FUNCTION_BLOCK FB_CintaTransferirPale_SFC
VAR_INPUT
    // SFC-Flags
    SFCPause: BOOL;
    SFCReset: BOOL;
    
    // Indicadores de sincronizacion
    Ack: BOOL := TRUE;
    Execute: BOOL;
    
    // Parametros
    TpoCintaRetenedor: TIME := T#1S;
    TpoCintaSeparador: TIME := T#1S;
    TpoPaleSalida: TIME := T#1S;
    TpoPaleTransferencia: TIME := T#1S;
    
    // Entradas
    PalePresencia: BOOL;
END_VAR
VAR_OUTPUT
    // Indicadores de sincronizacion
    Done: BOOL;
    Ready: BOOL;
    // Salidas
    CintaMotorActiva: BOOL;
    CintaRetenedorBaja: BOOL;
    CintaSeparadorSube: BOOL;
END_VAR
VAR
END_VAR

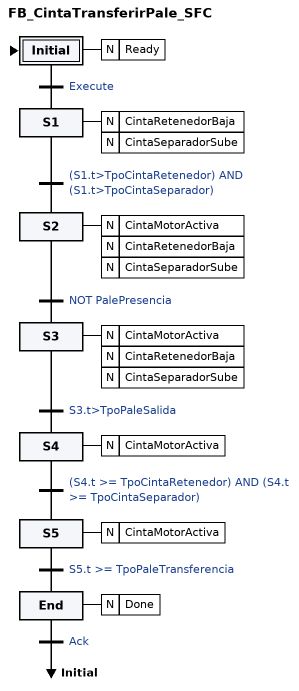
INITIAL_STEP Initial:
    Ready(N);
END_STEP
TRANSITION FROM Initial TO S1
    := Execute;
END_TRANSITION
STEP S1:
    CintaRetenedorBaja(N);
    CintaSeparadorSube(N);
END_STEP
TRANSITION FROM S1 TO S2
    := (S1.t>TpoCintaRetenedor) AND (S1.t>TpoCintaSeparador);
END_TRANSITION
STEP S2:
    CintaMotorActiva(N);
    CintaRetenedorBaja(N);
    CintaSeparadorSube(N);
END_STEP
TRANSITION FROM S2 TO S3
    := NOT PalePresencia;
END_TRANSITION
STEP S3:
    CintaMotorActiva(N);
    CintaRetenedorBaja(N);
    CintaSeparadorSube(N);
END_STEP
TRANSITION FROM S3 TO S4
    := S3.t>TpoPaleSalida;
END_TRANSITION
STEP S4:
    CintaMotorActiva(N);
END_STEP
TRANSITION FROM S4 TO S5
    := (S4.t >= TpoCintaRetenedor) AND (S4.t >= TpoCintaSeparador);
END_TRANSITION
STEP S5:
    CintaMotorActiva(N);
END_STEP
TRANSITION FROM S5 TO End
    := S5.t >= TpoPaleTransferencia;
END_TRANSITION
STEP End:
    Done(N);
END_STEP
TRANSITION FROM End TO Initial
    := Ack;
END_TRANSITION

END_FUNCTION_BLOCK

(* stored: Version 1.1.0.1, ProductVersion 3.1.4024.12
   POU FB_CintaTransferirPale_SFC: Id {f88ee7bd-e004-4fc2-9c9a-6c8228331871}, SpecialFunc None *)
